# B&R Automation Studio project MischeranlageRevA_Stufe03_DurchflussRegelung
Automation Studio 4.12.3.127 SP; technology packages: mappView 5.16.1

## Configuration Config1

CPU X20CP1382, AutomationRuntime E4.83, Build 4.1.2, Safety 0.0, Vc V4.72.5

### Task classes (Cpu.sw)
```
Cyclic#4:
  Simulation <- Simulation.prg
  Program <- Program.prg
Libraries: sys_lib, AsBrStr, runtime, Library
```

### Hardware
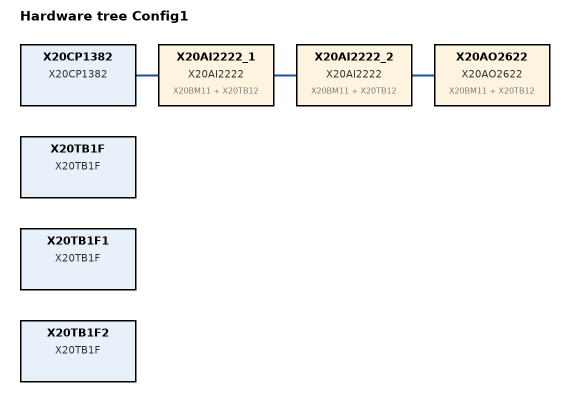
```
X20AI2222_1 : X20AI2222 v1.2.0.0  [SS1 -> X20TB12a.SS; SL -> X20BM11a.SL1]
X20AI2222_2 : X20AI2222 v1.2.0.0  [SS1 -> X20TB12.SS; SL -> X20BM11.SL1]
X20AO2622 : X20AO2622 v1.3.0.0  [SS1 -> X20TB12b.SS; SL -> X20BM11b.SL1]
X20BM11 : X20BM11 v1.1.0.0  [X2X1 -> X20BM11a.X2X2]
X20BM11a : X20BM11 v1.1.0.0  [X2X1 -> X20CP1382.IF6]
X20BM11b : X20BM11 v1.1.0.0  [X2X1 -> X20BM11.X2X2]
X20CP1382 : X20CP1382 v1.14.0.0  [X1 -> X1.SL; X2 -> X2.SL; X3 -> X3.SL]
  Module X1 (Type=X1, Virtual=true, Version=1.14.0.0)
    Connection (Connector=SS1, TargetModule=X20TB1F, TargetConnector=SS)
    Connection (Connector=SL, TargetModule=X20CP1382, TargetConnector=X1)
  Module X2 (Type=X2, Virtual=true, Version=1.14.0.0)
    Connection (Connector=SS1, TargetModule=X20TB1F1, TargetConnector=SS)
    Connection (Connector=SL, TargetModule=X20CP1382, TargetConnector=X2)
  Module X3 (Type=X3, Virtual=true, Version=1.14.0.0)
    Connection (Connector=SS1, TargetModule=X20TB1F2, TargetConnector=SS)
    Connection (Connector=SL, TargetModule=X20CP1382, TargetConnector=X3)
  Connector IF2:
    ActivateDevice = 1
    Mode = DHCP Server
    ActivateSnmp = 2
  ConfigurationID = X20CP1382_Config1
  Simulation = 1
  ActivateOpcUa = 1
  OpcUaInformationModels_PV_Version = 1
X20TB12 : X20TB12 v1.0.0.0
X20TB12a : X20TB12 v1.0.0.0
X20TB12b : X20TB12 v1.0.0.0
X20TB1F : X20TB1F v1.0.0.0
X20TB1F1 : X20TB1F v1.0.0.0
X20TB1F2 : X20TB1F v1.0.0.0
```

## Logical view

### Global.var - Globale Variablen
```iecst
VAR

    (* EINGAENGE *)
	iB_S1: BOOL := FALSE; (* Taster "Start" *)
	iB_S2: BOOL := FALSE; (* Taster "Automatikbetrieb" *)
	iB_S5: BOOL := FALSE; (* Endlagenschalter "Schieber Zu" *)
	iB_S6: BOOL := FALSE; (* Endlagenschalter "Schieber Auf" *)
	iB_B4: BOOL := FALSE; (* Lichtschranke "Schuettgut auf Band" *)

	iA_L1: INT  := 0; (* Ultraschallsensor Distanzmessung Silo 1 *)
	iA_L2: INT  := 0; (* Ultraschallsensor Distanzmessung Silo 2 *)

	iA_F3: INT  := 0; (* Durchflusssensor Wassereinspritzung *)

	iA_R1: INT	:= 0; (* Poti zur Sollwerteinstellung "Menge aus Silo 1" *)
	iA_R2: INT	:= 0; (* Poti zur Sollwerteinstellung "Menge aus Silo 2" *)

	(* AUSGAENGE *)
	qB_Q1_1: BOOL := FALSE; (* Motorschuetz Foerderschnecke 1 *)
	qB_Q2_1: BOOL := FALSE; (* Motorschuetz Foerderschnecke 2 *)
	qB_Q3_1: BOOL := FALSE; (* Motorschuetz Mischer *)
	qB_Q4_1: BOOL := FALSE; (* Motorschuetz Schieber auf *)
	qB_Q4_2: BOOL := FALSE; (* Motorschuetz Schieber zu *)
	qB_Q5_1: BOOL := FALSE; (* Motorschuetz Band *)

	qA_Y3: INT := 0; (* Regelventil Wassereinspritzung *)

	qB_P1: BOOL := FALSE; (* Meldeleuchte "Fuellstand zu gering" *)
	qB_P2: BOOL := FALSE; (* Meldeleuchte "Automatikbetrieb aktiv" *)

END_VAR

VAR CONSTANT

	(* Silogeometrie *)
	cA_H1: REAL := 20;
	cA_R0: REAL := 1.25;
	cA_R1: REAL := 6.25;
	cA_dR: REAL := cA_R1 - cA_R0;

	cA_H_Min: REAL := 5;

	(* Messkonstanten *)
	cA_k_s: REAL := 1 / 32767 * 99;

END_VAR
```

- Visualisation Logical/mappView (not shown)

### Library Logical/Library (IEC)

#### Library.fun - Exported functions and function blocks
```iecst
{REDUND_ERROR} FUNCTION VolumenImSilo : REAL (*Berechnung des Volumens im Silo in Abhängigkeit von h*) (*$GROUP=User,$CAT=User,$GROUPICON=User.png,$CATICON=User.png*)
	VAR_INPUT
		iA_h : REAL; (*Fuellhoehe*)
		iA_H1 : REAL; (*Hoehe Konus*)
		iA_R0 : REAL; (*Radius Konus*)
		iA_R1 : REAL; (*Radius Zylinder*)
	END_VAR
	VAR
		iA_dR : REAL; (*delta radius R1 - R0 vom Konus*)
		xA_V1 : REAL; (*Volumen 1 im Konus*)
		xA_V2 : REAL; (*Volumen 2 im Zylinder*)
	END_VAR
END_FUNCTION
```

#### VolumenImSilo.st
```iecst
(* Berechnung des Volumens im Silo in Abhängigkeit von h *)
FUNCTION VolumenImSilo
	iA_dR := iA_R1 - iA_R0;

	IF iA_h >= iA_H1 THEN
		xA_V1 := (iA_dR ** 2) / 3 + iA_dR * iA_R0 + (iA_R0 ** 2);
		xA_V1 := xA_V1 * 3.141 * iA_H1;

		xA_V2 := 3.141 * (iA_R1 ** 2) * (iA_h - iA_H1);
	ELSE
		xA_V1 := (iA_dR ** 2) / 3 / (iA_H1 ** 2) * iA_h;
		xA_V1 := (xA_V1 + iA_dR * iA_R0 / iA_H1) * iA_h;
		xA_V1 := (xA_V1 + (iA_R0 ** 2)) * iA_h * 3.141;

		xA_V2 := 0;
	END_IF;
	VolumenImSilo := xA_V1 + xA_V2;
END_FUNCTION
```

### Program Logical/Simulation (IEC)

#### Variables.var
```iecst
VAR

	(* Potentiometer *)
	xA_R1: REAL 	:= 0;
	xA_R2: REAL 	:= 0;
	tmpA_R1: REAL	:= 0;
	tmpA_R2: REAL	:= 0;

	(* Zustaende *)
	z_Auffahren: BOOL := FALSE;
	z_Zufahren:  BOOL := FALSE;

	(* Zeitvariablen *)
	xA_T_Schieber: INT := 0;
	xA_T_S1: INT := 0;
	xA_T_S2: INT := 0;

	(* Fuellstand Mischer *)
	xA_Mischer: REAL := 0;

	(* Silos *)
	xA_V1_1: REAL := 0;
	xA_V1_2: REAL := 0;
	xA_dV1:  REAL := 0;
	xA_A1:   REAL := 0;
	xA_h1:   REAL := 0;
	xA_dh1:  REAL := 0;

	xA_V2_1: REAL := 0;
	xA_V2_2: REAL := 0;
	xA_dV2:  REAL := 0;
	xA_A2:   REAL := 0;
	xA_h2:   REAL := 0;
	xA_dh2:  REAL := 0;

	xA_s1:   REAL := 0;
	xA_s2:   REAL := 0;

	(* Leitungsdruck *)
	xA_Druck: 			REAL := 5.0;
	xA_SteigenderDruck: REAL := 0.3;
	xA_FallenderDruck: 	REAL := 0.15;
	xA_MinDruck: 		REAL := 3;
	xA_MaxDruck: 		REAL := 8;
	xB_DruckSteigt:		BOOL := FALSE;

	(* Leitungsdurchfluss *)
	xA_Fluss: 	REAL 	:= 0;
	xA_Y3_Sim: 	INT 	:= 0;
	xA_dY3: 	INT 	:= 1300;
	xA_HystY3:	INT		:= 320;

END_VAR

VAR CONSTANT

	(* Zeitkonstanten *)
	cA_T_Zykl: INT := 100;
	cA_T_Schieber: INT := 3000;
	cA_T_S1: INT := 500;
	cA_T_S2: INT := 500;

END_VAR
```

#### Main.st
```iecst
PROGRAM _INIT

    (* Nullen der Zeitvariablen *)
	xA_T_Schieber := 0;
	xA_T_S1 := 0;

	(* Silofuellstaende zu Beginn*)
	xA_h1 := 25;
	xA_h2 := 32;

	xA_A1 := 0;

END_PROGRAM

PROGRAM _CYCLIC

    (* Potentiometer *)

	IF xA_R1 > 250 THEN
		xA_R1 := 250;
	ELSIF xA_R1 < 10 THEN
		xA_R1 := 10;
	END_IF;

	IF xA_R2 > 250 THEN
		xA_R2 := 250;
	ELSIF xA_R2 < 10 THEN
		xA_R2 := 10;
	END_IF;

	tmpA_R1 := (xA_R1 - 10) / 240 * 32767 * 0.8;
	iA_R1 := REAL_TO_INT(tmpA_R1);
	tmpA_R2 := (xA_R2 - 10) / 240 * 32767 * 0.8;
	iA_R2 := REAL_TO_INT(tmpA_R2);

    (* Silo 1 *)

	IF qB_Q1_1 THEN
		xA_dV1 := 10 * cA_T_Zykl;
		xA_dV1 := xA_dV1 / 1000;
	ELSE
		xA_dV1 := 0;
	END_IF;

	IF xA_h1 < cA_H1 THEN
		xA_A1 := (cA_dR * xA_h1) / cA_H1 + cA_R0;
	ELSE
		xA_A1 := cA_R1;
	END_IF;

	xA_A1 := xA_A1 ** 2;
	xA_A1 := xA_A1 * 3.141;
	xA_dh1 := xA_dV1 / xA_A1;
	xA_h1 := xA_h1 - xA_dh1;

	IF xA_h1 < 0 THEN
		xA_h1 := 0;
	END_IF;

	xA_s1 := 40 - xA_h1;
	iA_L1 := REAL_TO_INT((xA_s1 - 1) / 99 * 32767);

	(* Silo 2 *)

	IF qB_Q2_1 THEN
		xA_dV2 := 10 * cA_T_Zykl;
		xA_dV2 := xA_dV2 / 1000;
	ELSE
		xA_dV2 := 0;
	END_IF;

	IF xA_h2 < cA_H1 THEN
		xA_A2 := (cA_dR * xA_h2) / cA_H1 + cA_R0;
	ELSE
		xA_A2 := cA_R1;
	END_IF;

	xA_A2 := xA_A2 ** 2;
	xA_A2 := xA_A2 * 3.141;
	xA_dh2 := xA_dV2 / xA_A2;
	xA_h2 := xA_h2 - xA_dh2;

	IF xA_h2 < 0 THEN
		xA_h2 := 0;
	END_IF;

	xA_s2 := 40 - xA_h2;
	iA_L2 := REAL_TO_INT((xA_s2 - 1) / 99 * 32767);

	(* Steuerung der Anlage *)

	(* Mischer befuellen *)
	IF qB_Q1_1 AND (xA_h1 > 0) THEN
		xA_Mischer := xA_Mischer + 1;
	END_IF;

	IF qB_Q2_1 AND (xA_h2 > 0) THEN
		xA_Mischer := xA_Mischer + 1;
	END_IF;

	IF xA_Mischer < 0 THEN
		xA_Mischer := 0;
	END_IF;

	(* Mischer entleeren *)
	IF xA_T_Schieber > 0 THEN
		xA_Mischer := xA_Mischer - 0.001 * xA_T_Schieber;
	END_IF;

	(* Paralleles Auf- und Zufahren unterbinden *)
	z_Auffahren := qB_Q4_1 AND NOT z_Zufahren  AND NOT iB_S6;
	z_Zufahren  := qB_Q4_2 AND NOT z_Auffahren AND NOT iB_S5;

	(* Laufzeit Schieber auffahren *)
	IF z_Auffahren THEN
		xA_T_Schieber := xA_T_Schieber + cA_T_Zykl;
	END_IF

	(* Laufzeit Schieber zufahren *)
	IF z_Zufahren THEN
		xA_T_Schieber := xA_T_Schieber - cA_T_Zykl;
	END_IF

	(* Erreichen der Schieberendlagen *)
	iB_S6 := (xA_T_Schieber >= cA_T_Schieber);
	iB_S5 := (xA_T_Schieber <= 0);

	(* Zeug faellt auf's Band solang Schieber offen und Mischer nicht leer *)
	iB_B4 := (xA_Mischer > 0) AND (xA_T_Schieber > cA_T_Schieber / 5);

	(* Taster zuruecksetzen *)
	IF iB_S1 THEN
		xA_T_S1 := xA_T_S1 + cA_T_Zykl;
	ELSE
		xA_T_S1 := 0;
	END_IF;

	iB_S1 := iB_S1 AND NOT (xA_T_S1 >= cA_T_S1);

	IF iB_S2 THEN
		xA_T_S2 := xA_T_S2 + cA_T_Zykl;
	ELSE
		xA_T_S2 := 0;
	END_IF;

	iB_S2 := iB_S2 AND NOT (xA_T_S2 >= cA_T_S2);

	(* Leitungsdruck *)
	IF xB_DruckSteigt THEN
		xA_Druck := xA_Druck + xA_SteigenderDruck * cA_T_Zykl / 1000;
		xB_DruckSteigt := (xA_Druck < xA_MaxDruck);
	ELSE
		xA_Druck := xA_Druck - xA_FallenderDruck * cA_T_Zykl / 1000;
		xB_DruckSteigt := (xA_Druck < xA_MinDruck);
	END_IF;

	(*Durchfluss*)
	(* alt
	IF qA_Y3 > xA_Y3_Sim + xA_HystY3 THEN
		xA_Y3_Sim := xA_Y3_Sim + xA_dY3;
	ELSIF qA_Y3 < xA_Y3_Sim - xA_HystY3 THEN
		xA_Y3_Sim := xA_Y3_Sim - xA_dY3;
	END_IF;
	*)

	(* Darstellung der Strecke als PT1 *)
	xA_Y3_Sim := REAL_TO_INT((qA_Y3 - xA_Y3_Sim) / 20 + xA_Y3_Sim);

	IF xA_Y3_Sim < 0 THEN
		xA_Y3_Sim := 0;
	END_IF;

	IF xA_Y3_Sim > 32000 THEN
		xA_Y3_Sim := 32000;
	END_IF;

	xA_Fluss := xA_Y3_Sim * xA_Druck * 0.47 / 32767;
	iA_F3 := REAL_TO_INT(xA_Fluss / 10 * 32767);

END_PROGRAM

PROGRAM _EXIT
    (* Insert code here *)

END_PROGRAM
```

### Program Logical/Program (IEC)

#### Main.st - Init, cyclic, exit code
```iecst
(*Zugriff auf Simulation über Webbrowser (Chrome oder EDGE) http://localhost:81/*)
PROGRAM _INIT

	(* Silos initialisieren *)
	typSilo_Silo1.iA_Dichte := 1;
	typSilo_Silo1.iA_dR		:= cA_dR;
	typSilo_Silo1.iA_H1		:= cA_H1;
	typSilo_Silo1.iA_H_Min	:= cA_H_Min;
	typSilo_Silo1.iA_R0		:= cA_R0;
	typSilo_Silo1.iA_R1		:= cA_R1;
	typSilo_Silo1.iB_Init	:= TRUE;

	typSilo_Silo2.iA_Dichte := 1;
	typSilo_Silo2.iA_dR		:= cA_dR;
	typSilo_Silo2.iA_H1		:= cA_H1;
	typSilo_Silo2.iA_H_Min	:= cA_H_Min;
	typSilo_Silo2.iA_R0		:= cA_R0;
	typSilo_Silo2.iA_R1		:= cA_R1;
	typSilo_Silo2.iB_Init	:= TRUE;

	(* Standard Mengensollwerte *)
	xA_SwMenge1 := 150;
	xA_SwMenge2 := 100;

	(* Durchflussregelung initialisieren *)
	typPiRegler_Durchflussregler.iA_SW := 3276;
	typPiRegler_Durchflussregler.iA_Kp := 6;
	typPiRegler_Durchflussregler.iA_Tp := 0.1;
	typPiRegler_Durchflussregler.iA_Tn := 0.5;
	typPiRegler_Durchflussregler.iA_dt := 0.1;
	typPiRegler_Durchflussregler.iA_yMax := 32700;
	typPiRegler_Durchflussregler.iA_yMin := 0;

END_PROGRAM

PROGRAM _CYCLIC

	(* Analogwerte skalieren *)
	xA_h1 := 40 - iA_L1 * cA_k_h1 - 1;
	xA_h2 := 40 - iA_L2 * cA_k_h2 - 1;
	xA_SwMenge1 := 240 * 1.25 * iA_R1 / 32767 + 10;
	xA_SwMenge2 := 240 * 1.25 * iA_R2 / 32767 + 10;

	(* Werte an Silos uebergeben und berechnen *)
	typSilo_Silo1.iA_h := xA_h1;
	typSilo_Silo2.iA_h := xA_h2;
	typSilo_Silo1.iA_SwMenge := xA_SwMenge1;
	typSilo_Silo2.iA_SwMenge := xA_SwMenge2;
	typSilo_Silo1();
	typSilo_Silo2();

	(* Pruefe Starttransition *)
	xB_T0 := iB_S1 AND z_0;
	xB_T0 := xB_T0 AND typSilo_Silo1.qB_Freigabe;
	xB_T0 := xB_T0 AND typSilo_Silo2.qB_Freigabe;

	xB_FehlerFuellstand1 := (iB_S1 OR xB_FehlerFuellstand1) AND NOT typSilo_Silo1.qB_Freigabe;
	xB_FehlerFuellstand2 := (iB_S1 OR xB_FehlerFuellstand2) AND NOT typSilo_Silo2.qB_Freigabe;

	(* Zustandskette *)
	z_6 := NOT iB_S5 AND (z_6 OR (z_4 AND NOT iB_B4)); (* Schieber zufahren *)
	z_5 := NOT xB_T5 AND (z_5 OR (z_4 AND NOT iB_B4)); (* Bandnachlaufzeit *)
	z_4 := NOT z_5   AND (z_4 OR (z_3 AND     iB_S6)); (* Abtransport *)
	z_3 := NOT z_4   AND (z_3 OR (z_2 AND     xB_T2)); (* Schieber auf und Abtransport *)
	z_2 := NOT z_3   AND (z_2 OR (z_1 AND     xB_T1)); (* Mischen *)
	z_1 := NOT z_2   AND (z_1 OR (z_0 AND     xB_T0)); (* Befuellen und Mischen *)
	z_0 := NOT (z_1 OR z_2 OR z_3 OR z_4 OR z_5 OR z_6);

	(* Befuellung *)
	xB_Befuelle1 := z_1 AND NOT (typSilo_Silo1.qA_AbgegebeneMenge >= xA_SwMenge1);
	xB_Befuelle2 := z_1 AND NOT (typSilo_Silo2.qA_AbgegebeneMenge >= xA_SwMenge2);
	xB_T1 := z_1 AND NOT (xB_Befuelle1 OR xB_Befuelle2);

	(* Zeitsteuerung *)
	IF z_2 THEN
		xA_T2 := xA_T2 + cA_T_Zykl;
	ELSE
		xA_T2 := 0;
	END_IF;

	IF z_5 THEN
		xA_T5 := xA_T5 + cA_T_Zykl;
	ELSE
		xA_T5 := 0;
	END_IF;

	(* xB_T1 := (xA_T1 >= cA_T1); *)
	xB_T2 := (xA_T2 >= cA_T2);
	xB_T5 := (xA_T5 >= cA_T5);

	(* Steuerung der Motor-Ausgaenge *)
	qB_Q1_1 := xB_Befuelle1;
	qB_Q2_1 := xB_Befuelle2;
	qB_Q3_1 := z_1 OR z_2;
	qB_Q4_1 := z_3;
	qB_Q4_2 := z_6;
	qB_Q5_1 := z_3 OR z_4 OR z_5;

	iA_L1 := iA_L1;
	iA_L2 := iA_L2;

	(* Mengenzaehler zuruecksetzen *)
	IF z_0 THEN
		typSilo_Silo1.iB_Reset := TRUE;
		typSilo_Silo2.iB_Reset := TRUE;
	END_IF

	(* P1 blinkt bei zu geringem Füllstand *)
	qB_P1 := (xB_FehlerFuellstand1 OR xB_FehlerFuellstand2) AND xB_T_Takt;

	xB_T_Takt := ((xA_T_Takt >= cA_T_Takt) OR xB_T_Takt) AND (xA_T_Takt > 0);

	IF xB_T_Takt THEN
		xA_T_Takt := xA_T_Takt - cA_T_Zykl;
	ELSE
		xA_T_Takt := xA_T_Takt + cA_T_Zykl;
	END_IF;

	(* Automatikbetrieb *)
	xB_S2_sF := iB_S2 AND NOT tmpB_S2; (* steigende Flanke an S2 *)
	xB_Auto := (NOT xB_S2_sF AND xB_Auto) OR (xB_S2_sF AND NOT xB_Auto);
	tmpB_S2 := iB_S2;
	qB_P2 := xB_Auto;
	iB_S1 := (z_0 AND xB_Auto) OR iB_S1;

	(* Durchflusstregelung *)
	typPiRegler_Durchflussregler.iB_Freigabe := z_2;
	typPiRegler_Durchflussregler.iA_IW := iA_F3;
	typPiRegler_Durchflussregler();
	qA_Y3 := REAL_TO_INT(typPiRegler_Durchflussregler.qA_y);

END_PROGRAM

PROGRAM _EXIT
	(* Insert code here *)

END_PROGRAM
```

#### Variables.var - Local variables
```iecst
(* Zustaende *)
VAR
	z_0 : BOOL := FALSE; (* Leerlauf *)
	z_1 : BOOL := FALSE; (* Befuellen und Mischen *)
	z_2 : BOOL := FALSE; (* Mischen *)
	z_3 : BOOL := FALSE; (* Schieber auffahren und Abtransport *)
	z_4 : BOOL := FALSE; (* Abtransport *)
	z_5 : BOOL := FALSE; (* Bandnachlaufzeit *)
	z_6 : BOOL := FALSE; (* Schieber zufahren *) (* Schalt- und Transitionsvariablen *)
	xB_T0 : BOOL := FALSE; (* Transition von z_0 nach z_1 *)
	xB_T1 : BOOL := FALSE; (* Transition von z_1 nach z_2 *)
	xB_Befuelle1 : BOOL := FALSE; (* Befuellung aus Silo 1 *)
	xB_Befuelle2 : BOOL := FALSE; (* Befuellung aus Silo 2 *)
	xB_FehlerFuellstand1 : BOOL := FALSE; (* Fehlermeldung Visu wg Fuellstand 1 *)
	xB_FehlerFuellstand2 : BOOL := FALSE; (* Fehlermeldung Visu wg Fuellstand 1 *)
	xB_S2_sF : BOOL := FALSE; (* steigende Flanke an S2 *)
	xB_Auto : BOOL := FALSE; (* Automatikbetrieb aktiv *) (* Zeitvariablen *)
	xA_T1 : INT := 0; (* Zeitmessung im z_1 *)
	xA_T2 : INT := 0; (* Zeitmessung im z_2 *)
	xA_T5 : INT := 0; (* Zeitmessung im z_5 *)
	xA_T_Takt : INT := 0; (* Zeitmessung Taktgeber *)
	xB_T2 : BOOL := FALSE; (* Weiterschaltzeitpunkt erreicht *)
	xB_T5 : BOOL := FALSE; (* Weiterschaltzeitpunkt erreicht *)
	xB_T_Takt : BOOL := FALSE; (* Schaltausgang Taktgeber *) (* Silos *)
	typSilo_Silo1 : Silo; (* Funktionsbaustein Silo 1 *)
	typSilo_Silo2 : Silo; (* Funktionsbaustein Silo 2 *)
	xA_h1 : REAL := 0; (* Errechnete Fuellhoehe Silo 1 *)
	xA_h2 : REAL := 0; (* Errechnete Fuellhoehe Silo 2 *)
	xA_SwMenge1 : REAL := 0; (* Sollwert der abzuwiegenden Menge aus Silo 1 *)
	xA_SwMenge2 : REAL := 0; (* Sollwert der abzuwiegenden Menge aus Silo 2 *) (* "temporaere" Variablen *)
	tmpB_S2 : BOOL := FALSE; (* Letzter Zustand von Taster S2 *) (* Durchflussregelung *)
	typPiRegler_Durchflussregler : PiRegler;
END_VAR
(* Zeitkonstanten *)
VAR CONSTANT
	cA_T1 : INT := 10000; (* Befuellzeit *)
	cA_T2 : INT := 20000; (* Mischernachlaufzeit *)
	cA_T5 : INT := 5000; (* Bandnachlaufzeit *)
	cA_T_Takt : INT := 500; (* Taktzeit / 2 *)
	cA_T_Zykl : INT := 100; (* Umrechnungskonstanten Analogwerte *)
	cA_k_h1 : REAL := 99 / 32767;
	cA_k_h2 : REAL := 99 / 32767;
END_VAR
```

#### LocalFunctions.fun
```iecst
{REDUND_ERROR} FUNCTION_BLOCK Silo (*TODO: Hier einen Kommentar eingeben*) (*$GROUP=User,$CAT=User,$GROUPICON=User.png,$CATICON=User.png*)
	VAR_INPUT
		iA_h : REAL;
		iA_SwMenge : REAL;
		iB_Init : BOOL;
		iB_Reset : BOOL;
		iA_H1 : REAL;
		iA_R0 : REAL;
		iA_R1 : REAL;
		iA_Dichte : REAL;
		qB_SwErreicht : BOOL;
		iA_dR : REAL;
		iA_H_Min : REAL;
	END_VAR
	VAR_OUTPUT
		qB_Freigabe : BOOL;
		qA_MengeImSilo : REAL;
		qA_AbgegebeneMenge : REAL;
	END_VAR
	VAR
		xA_A : REAL;
		xA_h_zuletzt : REAL;
		xA_dh : REAL;
		xA_V1 : REAL;
		xA_V2 : REAL;
		xA_h : REAL;
		xA_Mindestfuellmenge : REAL;
		xA_dV : REAL;
	END_VAR
END_FUNCTION_BLOCK

{REDUND_ERROR} {REDUND_UNREPLICABLE} FUNCTION_BLOCK PiRegler (*TODO: Hier einen Kommentar eingeben*) (*$GROUP=User,$CAT=User,$GROUPICON=User.png,$CATICON=User.png*)
	VAR_INPUT
		iB_Freigabe: BOOL;
		iA_SW:       REAL;
		iA_IW:       REAL;
		iA_Kp:       REAL;
		iA_Tp:       REAL;
		iA_Tn:       REAL;
		iA_dt:       REAL;
		iA_yMin:     REAL;
		iA_yMax:     REAL;
	END_VAR

	VAR
		xB_AWU: BOOL;
		xA_u:   REAL;
		xA_yP1: REAL;
		xA_yP2: REAL;
		xA_yI:  REAL;
	END_VAR

	VAR_OUTPUT
		qA_y: REAL;
	END_VAR

END_FUNCTION_BLOCK
```

#### Silo.st
```iecst
(* TODO: Hier einen Kommentar eingeben *)
FUNCTION_BLOCK Silo

	(* Initialisierung *)
	IF iB_Init THEN

		(* Bestimmung der Mindestmenge im Silo *)
		xA_Mindestfuellmenge := VolumenImSilo(iA_H_Min, iA_H1, iA_R0, iA_R1) * iA_Dichte;

		iB_Init := FALSE;
		iB_Reset := TRUE;
	END_IF;

	(* Berechnungen bei Aenderung der Fuellhoehe *)
	IF (iA_h <> xA_h_zuletzt) THEN

		(* Ermittle Hoehendifferenz *)
		xA_dh := xA_h_zuletzt - iA_h;

		(* Bestimmung der Kreisflaeche anhand der Fuellhoehe *)
		IF iA_h < iA_H1 THEN
			xA_A := (iA_dR * iA_h) / iA_H1 + iA_R0;
		ELSE
			xA_A := iA_R1;
		END_IF;

		xA_A := xA_A ** 2;
		xA_A := xA_A * 3.141;

		(* Ermittle Volumenunterschied *)
		xA_dV := xA_A * xA_dh;

		(* Summiere abgegebene Menge auf *)
		qA_AbgegebeneMenge := qA_AbgegebeneMenge + xA_dV;

		(* Speichere aktuelle Fuellhoehe *)
		xA_h_zuletzt := iA_h;

	ELSE

		(* Keine Volumenaenderung ohne Hoehenaenderung *)
		xA_dV := 0;

	END_IF;

	(* Bestimmung der Menge im Silo *)
	qA_MengeImSilo := VolumenImSilo(iA_h, iA_H1, iA_R0, iA_R1) * iA_Dichte;

	(* Pruefe ob Sollwert erreicht *)
	IF qA_AbgegebeneMenge >= iA_SwMenge THEN
		qB_SwErreicht := TRUE;
	ELSE
		qB_SwErreicht := FALSE;
	END_IF;

	(* Pruefe ob Silo ausreichend voll *)
	IF qA_MengeImSilo - iA_SwMenge - xA_Mindestfuellmenge > 0 THEN
		qB_Freigabe := TRUE;
	ELSE
		qB_Freigabe := FALSE;
	END_IF;

	(* Zuruecksetzen *)
	IF iB_Reset THEN
		qA_AbgegebeneMenge := 0;
		iB_Reset := FALSE;
	END_IF;

END_FUNCTION_BLOCK
```

#### PiRegler.st
```iecst
(* TODO: Hier einen Kommentar eingeben *)
FUNCTION_BLOCK PiRegler

	IF iB_Freigabe THEN

		(* Bestimme Regeldifferenz *)
		xA_u := iA_SW - iA_IW;

		(* Berechne Proportionalanteil *)
		xA_yP1 := xA_u * iA_Kp;
		xA_yP2 := (xA_yP1 - xA_yP2) * iA_dt / iA_Tp + xA_yP2;

		(* Pruefe ob Aussteuerungsgrenze ueberschritten wird *)
		(* Falls ja, setze AntiWindUp(AWU)-Flag *)
		xB_AWU :=  (xA_yP1 < 0) AND (qA_y < iA_yMin);
		xB_AWU := ((xA_yP1 > 0) AND (qA_y > iA_yMax)) OR xB_AWU;

		(* Falls AWU-Flag inaktiv, berechne I-Anteil *)
		IF NOT xB_AWU THEN
			xA_yI := xA_yI + xA_yP1 / iA_Tn * iA_dt;
		END_IF;

		(* Addiere P- und I-Anteil --> Reglerausgangswert *)
		qA_y := xA_yP2 + xA_yI;

		IF qA_y > iA_yMax THEN
			qA_y := iA_yMax;
		END_IF;

		IF qA_y < iA_yMin THEN
			qA_y := iA_yMin;
		END_IF;

  	ELSE

		(* Falls keine Reglerfreigabe, setze alles zurueck *)
		xA_yP1 := 0;
		xA_yP2 := 0;
		xA_yI  := 0;
		qA_y   := 0;

	END_IF;

END_FUNCTION_BLOCK
```

Listed in the project but not available here: Logical/Global.typ, Logical/Libraries, Logical/Library/Types.typ, Logical/Library/Constants.var, Logical/Program/Types.typ
